Staubli VAL3: socketServer.dtx

bool bClawClosed = true
bool bDetectInput
bool bParseResult = true
jointRx home = {j1=0.299277, j2=90.551723, j3=0.116241, j4=-0.513613, j5=0.611835, j6=-177.732323}
jointRx homePoint = {j2=35, j6=-179}
jointRx jTest
jointRx joint1Test = {j2=3.0286646, j3=-0.380119, j4=-86.65991, j5=4.31054, j6=-179.150356}
jointRx joint1TestCopy = {j2=3.0286646, j3=-0.380119, j4=-86.65991, j5=4.31054, j6=-179.150356}
jointRx startPoint = {j2=29.71527, j3=59.600259, j4=-86.849417, j5=2.295044, j6=-178.473868}
jointRx waveIn = {j1=1.950737, j2=29.71527, j3=-3.0442775, j4=-86.849417, j5=2.295044, j6=-178.473868}
jointRx wristDown = {j1=1.747969, j2=68.569512, j3=20.407078, j4=-4.314453, j5=62.758443, j6=-270}
jointRx wristUp = {j1=1.747969, j2=68.569512, j3=20.407078, j4=-7.419285, j5=-49.114677, j6=-260.995824}
mdesc nom_speed = {rmax=9999, blend=off}
num nBuffer
num nFailCounter
num nIParseMovement
num nMovementData[3]
num nNum = -1
num nRXMovement = 70
num nTrsfJointArray[6]
  [0] = 11
  [1] = 3.0286646
  [2] = -0.380119
  [3] = -86.65991
  [4] = 4.31054
  [5] = -179.150356
num nXMovement = 11
num nZMovement = 168
pointRs pPointRs = {fatherId=world[0]}
pointRs pPointRs1 = {fatherId=world[0]}
sio sioSocket = {link=Socket\HelloServer}
string sBuffer
string sGetMovement
string sInput[50]
string sString = ")"
tool tClaw = {z=90, fatherId=flange[0], ioLink=valve1}
trsf trWorkingPoint
jointRx jJointRx = {j1=0.299277, j2=90.551723, j3=0.116241, j4=-0.513613, j5=0.611835, j6=-177.732323}
jointRx jJointRx1 = {j2=88.351928, j6=-179.151046}
jointRx homePointCopy = {j2=35, j6=-179}
num homePointArray[6]
  [1] = 35
  [5] = -179
